TYPE ST_VGC_NO EXTENDS ST_VGC :
STRUCT
	(* A normally open gate valve needs permission to close! *)
	(* EPICS Controls *)
	xCLS_SW	:	BOOL;
	xOvrdCls	:	BOOL;
	
	(* Interlocks *)
	xCLS_OK	:	BOOL;
	
	(* IO Controls *)
	xCLS_DO	:	BOOL;
	
	
END_STRUCT
END_TYPE

(* stored: Version 1.1.0.1, ProductVersion 3.1.4018.5
   DUT ST_VGC_NO: Id {637d6f45-b7b8-44fa-9c81-960a50d66588} *)
